(* IEC 61131-3 sources: IEC-63313-ST-Simulator/grammar/src/test/resources/iec61131_structuredtext, 20 files *)

(* ---- type.st ---- *)
TYPE ST_CAN_RXTX :
STRUCT
	uiTXCounter				:	UINT;
	uiRxCounter				:	UINT;
	uiNoOfRxTxMessages		:	UINT;
//	ar_stRxTxMessage		:	ARRAY[0..9] OF ST_CAN_RXTX_MESSAGE;
END_STRUCT;
END_TYPE

TYPE ST_CAN_RXTX_MESSAGE :
STRUCT
	uiLength		:	UINT;
	udCobId			:	UDINT;
//	ar_usiData		:	ARRAY[0..7] OF USINT;
END_STRUCT;
END_TYPE

TYPE ST_GezeFTV :
STRUCT
	bEntriegelt					:	BOOL;
	bVerriegelt					:	BOOL;
	bRunAlarm					:	BOOL;
	bTuerZu						:	BOOL;	// 1/4
	bRueckmeldungVerriegelung	:	BOOL;	// 1/7
	bTuerAlarmZentrale			:	BOOL;	// 2/2
	bKurzzeitfreigabe			:	BOOL;
END_STRUCT;
END_TYPE

(* ---- type_bool_struct.st ---- *)
TYPE
  S_FA_STATUS : STRUCT
    BART_Hand : BOOL := TRUE;
    BART_Auto : BOOL := FALSE;
    Stoerung : BOOL := FALSE;
    Stoer_Quit : BOOL := FALSE;
    NotHalt : BOOL := FALSE;
    Takt : BOOL := FALSE;
  END_STRUCT;
END_TYPE

(* ---- interface.st ---- *)
INTERFACE I_Subject

METHOD Attach : BOOL
VAR_INPUT
	ipObserver		: I_Observer;
END_VAR

METHOD Detach : BOOL
VAR_INPUT
	ipObserver		: I_Observer;
END_VAR

(* ---- function_selection.st ---- *)
FUNCTION SEL : ANY (* binary selection *)
  VAR_INPUT
    G : BOOL;
    IN0 : ANY;
    IN1 : ANY;
  END_VAR
  IF G = 0 THEN
    SEL := IN0; (* selection of upper input *)
  ELSE
    SEL := IN1; (*selection of lower input *)
  END_IF;
END_FUNCTION

(* ---- function_block.st ---- *)
FUNCTION_BLOCK PUBLIC FB_Logger
VAR
  sFilenameExtension : STRING;
END_VAR

// A method starts with a declaration
METHOD PUBLIC Write : STRING
VAR_INPUT
  sMsg : STRING;
END_VAR

// A method declaration is followed by statements that form
// the method's body.
// The next method declaration implicitly terminates the
// preceding method's body!
IF G = 0 THEN
	SEL := 1;
ELSE
	SEL := 2;
END_IF;

/*
sMsg := CONCAT('logger: ', sMsg);
IF (sFilenameExtension = 'txt') THEN
  Write := WriteTxt(sMsg);
ELSIF (sFilenameExtension = 'csv') THEN
  Write := WriteCsv(sMsg);
ELSIF (sFilenameExtension = 'xml') THEN
  Write := WriteXml(sMsg);
END_IF
*/

METHOD CreateErrorLogDB : BOOL
VAR_INPUT
    sDBName : T_MaxString;
END_VAR

CASE nState_CreateDB OF
    0:
    	stDBConfig.sServer := CONCAT(CONCAT(sDBPath, sDBName), '.sdf');
    	stDBConfig.bAuthentification := FALSE;

    	nState_CreateDB := 1;
    1:
        IF fbPLCDBCreate.Database(pDatabaseConfig:= ADR(stDBConfig),
            cbDatabaseConfig:= SIZEOF(stDBConfig),
            bCreateXMLConfig:= FALSE,
            pDBID:= 0) THEN
            ipResultEvt := fbPLCDBCreate.ipTcResult;
            IF fbPLCDBCreate.bError THEN
                nState_CreateDB := 100;
            ELSE
                nState_CreateDB := 2;
            END_IF;
        END_IF;
     2:
        IF fbConfigTcDBSrv.Create(pTcDBSrvConfig:= ADR(stDBConfig),
            cbTcDBSrvConfig:= SIZEOF(stDBConfig), bTemporary:= TRUE,
             pConfigID:= ADR(nDBID) ) THEN
            ipResultEvt := fbConfigTcDBSrv.ipTcResult;
            IF fbConfigTcDBSrv.bError THEN
                nState_CreateDB := 100;
            ELSE
                nState_CreateDB := 3;
            END_IF;
        END_IF;
     3:
     	arrTableColumns[0].sName := 'ID';
        arrTableColumns[0].eType := E_ColumnType.BigInt;
        arrTableColumns[0].nLength := 8;
        arrTableColumns[0].sProperty := 'IDENTITY(1,1)';

        arrTableColumns[1].sName := 'Timestamp';
        arrTableColumns[1].eType := E_ColumnType.DateTime;
        arrTableColumns[1].nLength := 4;

        arrTableColumns[2].sName := 'Severity';
        arrTableColumns[2].eType := E_ColumnType.NVarChar;
        arrTableColumns[2].nLength := 10;

        arrTableColumns[3].sName := 'ErrorCode';
        arrTableColumns[3].eType := E_ColumnType.Integer;
        arrTableColumns[3].nLength := 4;

        arrTableColumns[4].sName := 'Message';
        arrTableColumns[4].eType := E_ColumnType.NVarChar;
        arrTableColumns[4].nLength := 255;

        IF fbPLCDBCreate.Table(hDBID:= nDBID, sTableName:= sTableName,
            pTableCfg:= ADR(arrTableColumns),
            cbTableCfg:= SIZEOF(arrTableColumns)) THEN
            ipResultEvt := fbPLCDBCreate.ipTcResultEvent;
            nState_CreateDB := 100;
        END_IF;
    100:
        IF _SetResultInfo(1033) THEN
            IF NOT bError THEN
                _bHasCreated := TRUE;
            END_IF;

            nState_CreateDB := 0;
        END_IF;
END_CASE;

END_FUNCTION_BLOCK

(* ---- function_block_inout_var.st ---- *)
FUNCTION_BLOCK FNC_BLK

  VAR_IN_OUT
    var_1 : BOOL;
    var_2 : BOOL;
  END_VAR

  VAR_INPUT
    var_3 : UINT;
    var_4 : UINT;
  END_VAR

END_FUNCTION_BLOCK

(* ---- function_block_simple.st ---- *)
FUNCTION_BLOCK FNC_BLK

  VAR_INPUT
    var_1 : BOOL;
  END_VAR

END_FUNCTION_BLOCK

(* ---- large_program.st ---- *)
/**/
TYPE
  S_FA_STATUS : STRUCT
    BART_Hand : BOOL := TRUE;
    BART_Auto : BOOL := FALSE;
    Stoerung : BOOL := FALSE;
    Stoer_Quit : BOOL := FALSE;
    NotHalt : BOOL := FALSE;
    Takt : BOOL := FALSE;
  END_STRUCT;
END_TYPE

FUNCTION_BLOCK AKT_5_2_MV
  VAR_INPUT
    status : S_FA_STATUS;
    Hand_P1 : BOOL;
    Hand_P2 : BOOL;
  END_VAR
  VAR_INPUT
    SEN_P1 : BOOL;
    SEN_P2 : BOOL;
  END_VAR

  VAR_OUTPUT
    s_MV_P2_FF : BOOL;
  END_VAR

  VAR
    SR0 : SR;
  END_VAR
  VAR
    DebugBoolean : BOOL;
    TON0 : TON;
  END_VAR

  VAR CONSTANT
    const_T_Laufzeit_P2 : TIME := T#10s;
  END_VAR

  VAR
    _TMP_AND6_OUT : BOOL;
    _TMP_AND9_OUT : BOOL;
    _TMP_NOT17_OUT : BOOL;
    _TMP_AND15_OUT : BOOL;
  END_VAR

  // compute the control input for Magnetventil Position 2 using a Reset-dominant flip flop
  // and store the result into the out parameter s_MV_P2_FF
  _TMP_AND6_OUT := AND(status.BART_Hand, Hand_P2);
  _TMP_AND9_OUT := AND(status.BART_Hand, Hand_P1);
  SR0(S1 := _TMP_AND6_OUT, R := _TMP_AND9_OUT);
  s_MV_P2_FF := SR0.Q1;

  // Error detection - Laufzeitueberwachung towards Magnetventil Position 2
  _TMP_NOT17_OUT := NOT(SEN_P2);
  _TMP_AND15_OUT := AND(_TMP_NOT17_OUT, Hand_P2);
  TON0(IN := _TMP_AND15_OUT, PT := const_T_Laufzeit_P2);
  DebugBoolean := TON0.Q;

END_FUNCTION_BLOCK

/* We cannot parse functions yet!
FUNCTION FA_SERV : BOOL
  VAR_INPUT
    status : S_FA_STATUS;
    BART_Hand : BOOL;
    BART_Auto : BOOL;
    Stoerung : BOOL;
    Stoer_Quit : BOOL;
    NotHalt : BOOL;
  END_VAR

  status.BART_Hand := BART_Hand;
  status.BART_Auto := BART_Auto;
  status.Stoerung := Stoerung;
  status.Stoer_Quit := Stoer_Quit;
  status.NotHalt := NotHalt;

  FA_SERV := status.BART_Hand;
END_FUNCTION
*/

PROGRAM program0_POU
  VAR
    FA_Start_T_HMI : BOOL;
    FA_Init_T_HMI : BOOL;
    FA_Sonder_T_HMI : BOOL;
    FA_Stop_T_HMI : BOOL;
    FA_BART_Hand_T_HMI : BOOL := TRUE;
    FA_BART_Auto_T_HMI : BOOL;
    FA_BART_Auto_Einzel_T_HMI : BOOL;
    FA_Stoerung_T_HMI : BOOL;
    FA_Stoer_Quit_T_HMI : BOOL;
    FA_NotHalt_T_HMI : BOOL;
    DebugBoolean : BOOL;
  END_VAR
  VAR_EXTERNAL
    global_status : S_FA_STATUS;
  END_VAR
  VAR
    AKT_5_2_MV0 : AKT_5_2_MV;
    Zyl1_T_P1_HMI : BOOL;
    //Zyl1_T_P2_HMI : BOOL := TRUE;
    Zyl1_T_P2_HMI : BOOL := FALSE;
    //Zyl1_T_P2_HMI : BOOL;
    s_MV_P2_FF : BOOL;
    SEN_P1_T_HMI : BOOL := TRUE;
    SEN_P2_T_HMI : BOOL := FALSE;
    _TMP_FA_SERV1_OUT : BOOL;
  END_VAR

  global_status.BART_Hand := FA_BART_Hand_T_HMI;

  //_TMP_FA_SERV1_OUT := FA_SERV(global_status, FA_BART_Hand_T_HMI, FA_BART_Auto_T_HMI, FA_Stoerung_T_HMI, FA_Stoer_Quit_T_HMI, FA_NotHalt_T_HMI);

  DebugBoolean := _TMP_FA_SERV1_OUT;

  AKT_5_2_MV0(
    status := global_status,
    Hand_P1 := Zyl1_T_P1_HMI,
    Hand_P2 := Zyl1_T_P2_HMI,
    SEN_P1 := SEN_P1_T_HMI,
    SEN_P2 := SEN_P2_T_HMI
  );

  s_MV_P2_FF := AKT_5_2_MV0.s_MV_P2_FF;

END_PROGRAM

FUNCTION_BLOCK FA
  VAR
    Status : S_FA_STATUS;
  END_VAR

  Status.Stoerung := TRUE;
END_FUNCTION_BLOCK

/*
FUNCTION_BLOCK SequenctialFunctionChart
  VAR
    RedLight : BOOL;
    OrangeLight : BOOL;
    GreenLight : BOOL;
    Step_0_Active : BOOL := TRUE;
    Step_1_Active : BOOL := FALSE;
    Step_2_Active : BOOL := FALSE;
    TON0 : TON;
    TON1 : TON;
    TON2 : TON;
  END_VAR

  INITIAL_STEP Step0:
    RedLight(N);
    Step_0_Active(N);
    COMPUTE_FUNCTION_BLOCKS(S);
  END_STEP

  ACTION COMPUTE_FUNCTION_BLOCKS:
    TON0(IN := Step_0_Active, PT := T#6s);
    TON1(IN := Step_1_Active, PT := T#6s);
    TON2(IN := Step_2_Active, PT := T#6s);
  END_ACTION

  TRANSITION FROM Step0 TO Step1
    := TON0.Q;
  END_TRANSITION

  STEP Step1:
    GreenLight(N);
    Step_1_Active(N);
  END_STEP

  TRANSITION FROM Step1 TO Step2
    := TON1.Q;
  END_TRANSITION

  STEP Step2:
    OrangeLight(N);
    Step_2_Active(N);
  END_STEP

  TRANSITION FROM Step2 TO Step0
    := TON2.Q;
  END_TRANSITION

END_FUNCTION_BLOCK
*/

CONFIGURATION Config0

  RESOURCE Res0 ON PLC
    VAR_GLOBAL
      global_status : S_FA_STATUS;
    END_VAR
    TASK task0(INTERVAL := T#20ms,PRIORITY := 0);
    PROGRAM instance0 WITH task0 : program0_POU;
  END_RESOURCE

END_CONFIGURATION

(* ---- large_program_2.st ---- *)
TYPE
  S_FA_STATUS : STRUCT
    BART_Hand : BOOL := TRUE;
    BART_Auto : BOOL := FALSE;
    Stoerung : BOOL := FALSE;
    Stoer_Quit : BOOL := FALSE;
    NotHalt : BOOL := FALSE;
    Takt : BOOL := FALSE;
  END_STRUCT;
END_TYPE

FUNCTION_BLOCK AKT_5_2_MV
    /**/
  VAR_IN_OUT
    status : S_FA_STATUS;
  END_VAR

  VAR_INPUT
    //status : S_FA_STATUS;
    Hand_P1 : BOOL;
    Hand_P2 : BOOL;
  END_VAR
  VAR
    SR0 : SR;
  END_VAR
  VAR_OUTPUT
    s_MV_P2_FF : BOOL;
  END_VAR
  VAR
    DebugBoolean : BOOL;
    TON0 : TON;
  END_VAR
  VAR CONSTANT
    const_T_Laufzeit_P2 : TIME := T#10s;
  END_VAR
  VAR_INPUT
    SEN_P1 : BOOL;
    SEN_P2 : BOOL;
  END_VAR
  VAR
    _TMP_AND6_OUT : BOOL;
    _TMP_AND9_OUT : BOOL;
    _TMP_NOT17_OUT : BOOL;
    _TMP_AND15_OUT : BOOL;
  END_VAR

  _TMP_AND6_OUT := AND(status.BART_Hand, Hand_P2);
  _TMP_AND9_OUT := AND(status.BART_Hand, Hand_P1);
  SR0(S1 := _TMP_AND6_OUT, R := _TMP_AND9_OUT);
  s_MV_P2_FF := SR0.Q1;
  _TMP_NOT17_OUT := NOT(SEN_P2);
  _TMP_AND15_OUT := AND(_TMP_NOT17_OUT, Hand_P2);
  TON0(IN := _TMP_AND15_OUT, PT := const_T_Laufzeit_P2);
  status.Stoerung := TON0.Q;
END_FUNCTION_BLOCK

/*
FUNCTION FA_SERV : BOOL
  VAR_INPUT
    status : S_FA_STATUS;
    BART_Hand : BOOL;
    BART_Auto : BOOL;
    Stoerung : BOOL;
    Stoer_Quit : BOOL;
    NotHalt : BOOL;
  END_VAR

  status.BART_Hand := BART_Hand;
  FA_SERV := status.BART_Hand;
  status.BART_Auto := BART_Auto;
  status.Stoerung := Stoerung;
  status.Stoer_Quit := Stoer_Quit;
  status.NotHalt := NotHalt;
END_FUNCTION
*/

PROGRAM program0_POU
  VAR
    FA_Start_T_HMI : BOOL;
    FA_Init_T_HMI : BOOL;
    FA_Sonder_T_HMI : BOOL;
    FA_Stop_T_HMI : BOOL;
    FA_BART_Hand_T_HMI : BOOL := TRUE;
    FA_BART_Auto_T_HMI : BOOL;
    FA_BART_Auto_Einzel_T_HMI : BOOL;
    FA_Stoerung_T_HMI : BOOL;
    FA_Stoer_Quit_T_HMI : BOOL;
    FA_NotHalt_T_HMI : BOOL;
    DebugBoolean : BOOL;
  END_VAR
  VAR_EXTERNAL
    global_status : S_FA_STATUS;
  END_VAR
  VAR
    AKT_5_2_MV0 : AKT_5_2_MV;
    Zyl1_T_P1_HMI : BOOL;
    Zyl1_T_P2_HMI : BOOL;
    s_MV_P2_FF : BOOL;
    SEN_P1_T_HMI : BOOL := TRUE;
    SEN_P2_T_HMI : BOOL := FALSE;
    _TMP_FA_SERV1_OUT : BOOL;
  END_VAR

  global_status.BART_Hand := FA_BART_Hand_T_HMI;
  //_TMP_FA_SERV1_OUT := FA_SERV(global_status, FA_BART_Hand_T_HMI, FA_BART_Auto_T_HMI, FA_Stoerung_T_HMI, FA_Stoer_Quit_T_HMI, FA_NotHalt_T_HMI);
  DebugBoolean := _TMP_FA_SERV1_OUT;
  AKT_5_2_MV0(status := global_status, Hand_P1 := Zyl1_T_P1_HMI, Hand_P2 := Zyl1_T_P2_HMI, SEN_P1 := SEN_P1_T_HMI, SEN_P2 := SEN_P2_T_HMI);
  s_MV_P2_FF := AKT_5_2_MV0.s_MV_P2_FF;
END_PROGRAM

FUNCTION_BLOCK FA
  VAR
    Status : S_FA_STATUS;
  END_VAR

  Status.Stoerung := TRUE;
END_FUNCTION_BLOCK

/*
FUNCTION_BLOCK SequenctialFunctionChart
  VAR
    RedLight : BOOL;
    OrangeLight : BOOL;
    GreenLight : BOOL;
    Step_0_Active : BOOL := TRUE;
    Step_1_Active : BOOL := FALSE;
    Step_2_Active : BOOL := FALSE;
    TON0 : TON;
    TON1 : TON;
    TON2 : TON;
  END_VAR

  INITIAL_STEP Step0:
    RedLight(N);
    Step_0_Active(N);
    COMPUTE_FUNCTION_BLOCKS(S);
  END_STEP

  ACTION COMPUTE_FUNCTION_BLOCKS:
    TON0(IN := Step_0_Active, PT := T#6s);
    TON1(IN := Step_1_Active, PT := T#6s);
    TON2(IN := Step_2_Active, PT := T#6s);
  END_ACTION

  TRANSITION FROM Step0 TO Step1
    := TON0.Q;
  END_TRANSITION

  STEP Step1:
    GreenLight(N);
    Step_1_Active(N);
  END_STEP

  TRANSITION FROM Step1 TO Step2
    := TON1.Q;
  END_TRANSITION

  STEP Step2:
    OrangeLight(N);
    Step_2_Active(N);
  END_STEP

  TRANSITION FROM Step2 TO Step0
    := TON2.Q;
  END_TRANSITION

END_FUNCTION_BLOCK
*/

CONFIGURATION Config0

  RESOURCE Res0 ON PLC
    VAR_GLOBAL
      global_status : S_FA_STATUS;
    END_VAR
    TASK task0(INTERVAL := T#20ms,PRIORITY := 0);
    PROGRAM instance0 WITH task0 : program0_POU;
  END_RESOURCE
END_CONFIGURATION

(* ---- large_program_3.st ---- *)
TYPE
  S_FA_STATUS : STRUCT
    BART_Hand : BOOL := TRUE;
    BART_Auto : BOOL := FALSE;
    Stoerung : BOOL := FALSE;
    Stoer_Quit : BOOL := FALSE;
    NotHalt : BOOL := FALSE;
    Takt : BOOL := FALSE;
  END_STRUCT;
END_TYPE

FUNCTION_BLOCK AKT_5_2_MV
  VAR_IN_OUT
    status : S_FA_STATUS;
  END_VAR
  VAR_INPUT
    Hand_P1 : BOOL;
    Hand_P2 : BOOL;
  END_VAR
  VAR
    SR0 : SR;
  END_VAR
  VAR_OUTPUT
    s_MV_P2_FF : BOOL;
  END_VAR
  VAR
    DebugBoolean : BOOL;
    TON0 : TON;
  END_VAR
  VAR CONSTANT
    const_T_Laufzeit_P2 : TIME := T#10s;
  END_VAR
  VAR_INPUT
    SEN_P1 : BOOL;
    SEN_P2 : BOOL;
  END_VAR
  VAR
    RS0 : RS;
  END_VAR
  VAR_INPUT
    F_LZ_P2 : RS;
  END_VAR
  VAR_OUTPUT
    F_LZ_P3 : BOOL;
  END_VAR
  VAR
    _TMP_AND6_OUT : BOOL;
    _TMP_AND9_OUT : BOOL;
    _TMP_NOT17_OUT : BOOL;
    _TMP_AND15_OUT : BOOL;
  END_VAR

  _TMP_AND6_OUT := AND(status.BART_Hand, Hand_P2);
  _TMP_AND9_OUT := AND(status.BART_Hand, Hand_P1);
  SR0(S1 := _TMP_AND6_OUT, R := _TMP_AND9_OUT);
  s_MV_P2_FF := SR0.Q1;
  _TMP_NOT17_OUT := NOT(SEN_P2);
  _TMP_AND15_OUT := AND(_TMP_NOT17_OUT, Hand_P2);
  TON0(IN := _TMP_AND15_OUT, PT := const_T_Laufzeit_P2);
  RS0(S := TON0.Q);
  F_LZ_P3 := RS0.Q1;
END_FUNCTION_BLOCK
/*
FUNCTION FA_SERV : BOOL
  VAR_INPUT
    status : S_FA_STATUS;
    BART_Hand : BOOL;
    BART_Auto : BOOL;
    Stoerung : BOOL;
    Stoer_Quit : BOOL;
    NotHalt : BOOL;
  END_VAR

  status.BART_Hand := BART_Hand;
  FA_SERV := status.BART_Hand;
  status.BART_Auto := BART_Auto;
  status.Stoerung := Stoerung;
  status.Stoer_Quit := Stoer_Quit;
  status.NotHalt := NotHalt;
END_FUNCTION
*/
PROGRAM program0_POU
  VAR
    FA_Start_T_HMI : BOOL;
    FA_Init_T_HMI : BOOL;
    FA_Sonder_T_HMI : BOOL;
    FA_Stop_T_HMI : BOOL;
    FA_BART_Hand_T_HMI : BOOL := TRUE;
    FA_BART_Auto_T_HMI : BOOL;
    FA_BART_Auto_Einzel_T_HMI : BOOL;
    FA_Stoerung_T_HMI : BOOL;
    FA_Stoer_Quit_T_HMI : BOOL;
    FA_NotHalt_T_HMI : BOOL;
    DebugBoolean : BOOL;
  END_VAR
  VAR_EXTERNAL
    global_status : S_FA_STATUS;
  END_VAR
  VAR
    AKT_5_2_MV0 : AKT_5_2_MV;
    Zyl1_T_P1_HMI : BOOL;
    Zyl1_T_P2_HMI : BOOL;
    s_MV_P2_FF : BOOL;
    SEN_P1_T_HMI : BOOL := TRUE;
    SEN_P2_T_HMI : BOOL := FALSE;
    _TMP_FA_SERV1_OUT : BOOL;
  END_VAR

  global_status.BART_Hand := FA_BART_Hand_T_HMI;
  //_TMP_FA_SERV1_OUT := FA_SERV(global_status, FA_BART_Hand_T_HMI, FA_BART_Auto_T_HMI, FA_Stoerung_T_HMI, FA_Stoer_Quit_T_HMI, FA_NotHalt_T_HMI);
  DebugBoolean := _TMP_FA_SERV1_OUT;
  AKT_5_2_MV0(status := global_status, Hand_P1 := Zyl1_T_P1_HMI, Hand_P2 := Zyl1_T_P2_HMI, SEN_P1 := SEN_P1_T_HMI, SEN_P2 := SEN_P2_T_HMI);
  s_MV_P2_FF := AKT_5_2_MV0.s_MV_P2_FF;
END_PROGRAM

FUNCTION_BLOCK FA
  VAR
    Status : S_FA_STATUS;
  END_VAR

  Status.Stoerung := TRUE;
END_FUNCTION_BLOCK

/*
FUNCTION_BLOCK SequenctialFunctionChart
  VAR
    RedLight : BOOL;
    OrangeLight : BOOL;
    GreenLight : BOOL;
    Step_0_Active : BOOL := TRUE;
    Step_1_Active : BOOL := FALSE;
    Step_2_Active : BOOL := FALSE;
    TON0 : TON;
    TON1 : TON;
    TON2 : TON;
  END_VAR

  INITIAL_STEP Step0:
    RedLight(N);
    Step_0_Active(N);
    COMPUTE_FUNCTION_BLOCKS(S);
  END_STEP

  ACTION COMPUTE_FUNCTION_BLOCKS:
    TON0(IN := Step_0_Active, PT := T#6s);
    TON1(IN := Step_1_Active, PT := T#6s);
    TON2(IN := Step_2_Active, PT := T#6s);
  END_ACTION

  TRANSITION FROM Step0 TO Step1
    := TON0.Q;
  END_TRANSITION

  STEP Step1:
    GreenLight(N);
    Step_1_Active(N);
  END_STEP

  TRANSITION FROM Step1 TO Step2
    := TON1.Q;
  END_TRANSITION

  STEP Step2:
    OrangeLight(N);
    Step_2_Active(N);
  END_STEP

  TRANSITION FROM Step2 TO Step0
    := TON2.Q;
  END_TRANSITION

END_FUNCTION_BLOCK
*/

CONFIGURATION Config0

  RESOURCE Res0 ON PLC
    VAR_GLOBAL
      global_status : S_FA_STATUS;
    END_VAR
    TASK task0(INTERVAL := T#20ms,PRIORITY := 0);
    PROGRAM instance0 WITH task0 : program0_POU;
  END_RESOURCE
END_CONFIGURATION

(* ---- large_program_4.st ---- *)
TYPE
  S_FA_STATUS : STRUCT
    BART_Hand : BOOL := TRUE;
    BART_Auto : BOOL := FALSE;
    Stoerung : BOOL := FALSE;
    Stoer_Quit : BOOL := FALSE;
    NotHalt : BOOL := FALSE;
    Takt : BOOL := FALSE;
  END_STRUCT;
  Diag : STRUCT
    F_Paar_EN : BOOL := TRUE;
    F_LZ_P1_EN : BOOL := TRUE;
    F_LZ_P2_EN : BOOL := TRUE;
    F_LZ_P1_Zeit : TIME;
    F_LZ_P2_Zeit : TIME;
    Stoerung : BOOL := FALSE;
  END_STRUCT;
END_TYPE

FUNCTION_BLOCK AKT_5_2_MV
  VAR_IN_OUT
    status : S_FA_STATUS;
  END_VAR
  VAR_INPUT
    Hand_P1 : BOOL;
    Hand_P2 : BOOL;
  END_VAR
  VAR
    SR0 : SR;
    SR1 : SR;
  END_VAR
  VAR_OUTPUT
    s_MV_P1_FF : BOOL;
    s_MV_P2_FF : BOOL;
  END_VAR
  VAR
    DebugBoolean : BOOL;
    TON0 : TON;
    TON1 : TON;
  END_VAR
  VAR CONSTANT
    const_T_Laufzeit_P2 : TIME := T#10s;
  END_VAR
  VAR_INPUT
    SEN_P1 : BOOL;
    SEN_P2 : BOOL;
  END_VAR
  VAR
    RS0 : RS;
    RS1 : RS;
  END_VAR
  VAR_INPUT
    F_LZ_P2 : RS;
  END_VAR
  VAR_OUTPUT
    F_LZ_P3 : BOOL;
    F_LZ_P4 : BOOL;
  END_VAR
  VAR_IN_OUT
    Diag : Diag;
  END_VAR
  VAR
    _TMP_AND6_OUT : BOOL;
    _TMP_AND9_OUT : BOOL;
    _TMP_NOT17_OUT : BOOL;
    _TMP_AND15_OUT : BOOL;
    _TMP_OR30_OUT : BOOL;
    _TMP_NOT2_OUT : BOOL;
    _TMP_AND19_OUT : BOOL;
    _TMP_AND18_OUT : BOOL;
    _TMP_AND36_OUT : BOOL;
  END_VAR

  _TMP_AND6_OUT := AND(status.BART_Hand, Hand_P2);
  _TMP_AND9_OUT := AND(status.BART_Hand, Hand_P1);
  SR0(S1 := _TMP_AND6_OUT, R := _TMP_AND9_OUT);
  s_MV_P2_FF := SR0.Q1;

  _TMP_NOT17_OUT := NOT(SEN_P2);
  _TMP_AND15_OUT := AND(_TMP_NOT17_OUT, Hand_P2);
  TON0(IN := _TMP_AND15_OUT, PT := const_T_Laufzeit_P2);
  RS0(S := TON0.Q);

  _TMP_NOT2_OUT := NOT(SEN_P1);
  _TMP_AND19_OUT := AND(_TMP_NOT2_OUT, Hand_P1);
  TON1(IN := _TMP_AND19_OUT, PT := const_T_Laufzeit_P2);
  RS1(S := TON1.Q);

  F_LZ_P3 := RS0.Q1;
  _TMP_OR30_OUT := OR(F_LZ_P3, F_LZ_P4);
  Diag.Stoerung := _TMP_OR30_OUT;

  F_LZ_P4 := RS1.Q1;
  _TMP_AND18_OUT := AND(status.BART_Hand, Hand_P1);
  _TMP_AND36_OUT := AND(status.BART_Hand, Hand_P2);
  SR1(S1 := _TMP_AND18_OUT, R := _TMP_AND36_OUT);
  s_MV_P1_FF := SR1.Q1;

END_FUNCTION_BLOCK

/*
FUNCTION FA_SERV : BOOL
  VAR_INPUT
    status : S_FA_STATUS;
    BART_Hand : BOOL;
    BART_Auto : BOOL;
    Stoerung : BOOL;
    Stoer_Quit : BOOL;
    NotHalt : BOOL;
  END_VAR

  status.BART_Hand := BART_Hand;
  FA_SERV := status.BART_Hand;
  status.BART_Auto := BART_Auto;
  status.Stoerung := Stoerung;
  status.Stoer_Quit := Stoer_Quit;
  status.NotHalt := NotHalt;
END_FUNCTION
*/

PROGRAM program0_POU
  VAR
    FA_Start_T_HMI : BOOL;
    FA_Init_T_HMI : BOOL;
    FA_Sonder_T_HMI : BOOL;
    FA_Stop_T_HMI : BOOL;
    FA_BART_Hand_T_HMI : BOOL := TRUE;
    FA_BART_Auto_T_HMI : BOOL;
    FA_BART_Auto_Einzel_T_HMI : BOOL;
    FA_Stoerung_T_HMI : BOOL;
    FA_Stoer_Quit_T_HMI : BOOL;
    FA_NotHalt_T_HMI : BOOL;
    DebugBoolean : BOOL;
  END_VAR
  VAR_EXTERNAL
    global_status : S_FA_STATUS;
  END_VAR
  VAR
    AKT_5_2_MV0 : AKT_5_2_MV;
    Zyl1_T_P1_HMI : BOOL := FALSE;
    Zyl1_T_P2_HMI : BOOL := FALSE;
    s_MV_P2_FF : BOOL;
    SEN_P1_T_HMI : BOOL := TRUE;
    SEN_P2_T_HMI : BOOL := FALSE;
    Diag : Diag;
    _TMP_FA_SERV1_OUT : BOOL;
  END_VAR

  global_status.BART_Hand := FA_BART_Hand_T_HMI;
  //_TMP_FA_SERV1_OUT := FA_SERV(global_status, FA_BART_Hand_T_HMI, FA_BART_Auto_T_HMI, FA_Stoerung_T_HMI, FA_Stoer_Quit_T_HMI, FA_NotHalt_T_HMI);
  //DebugBoolean := _TMP_FA_SERV1_OUT;
  AKT_5_2_MV0(status := global_status, Hand_P1 := Zyl1_T_P1_HMI, Hand_P2 := Zyl1_T_P2_HMI, SEN_P1 := SEN_P1_T_HMI, SEN_P2 := SEN_P2_T_HMI, Diag := Diag);
  s_MV_P2_FF := AKT_5_2_MV0.s_MV_P2_FF;
END_PROGRAM

/*
FUNCTION_BLOCK FA
  VAR
    Status : S_FA_STATUS;
  END_VAR

  Status.Stoerung := TRUE;
END_FUNCTION_BLOCK

FUNCTION_BLOCK SequenctialFunctionChart
  VAR
    RedLight : BOOL;
    OrangeLight : BOOL;
    GreenLight : BOOL;
    Step_0_Active : BOOL := TRUE;
    Step_1_Active : BOOL := FALSE;
    Step_2_Active : BOOL := FALSE;
    TON0 : TON;
    TON1 : TON;
    TON2 : TON;
  END_VAR

  INITIAL_STEP Step0:
    RedLight(N);
    Step_0_Active(N);
    COMPUTE_FUNCTION_BLOCKS(S);
  END_STEP

  ACTION COMPUTE_FUNCTION_BLOCKS:
    TON0(IN := Step_0_Active, PT := T#6s);
    TON1(IN := Step_1_Active, PT := T#6s);
    TON2(IN := Step_2_Active, PT := T#6s);
  END_ACTION

  TRANSITION FROM Step0 TO Step1
    := TON0.Q;
  END_TRANSITION

  STEP Step1:
    GreenLight(N);
    Step_1_Active(N);
  END_STEP

  TRANSITION FROM Step1 TO Step2
    := TON1.Q;
  END_TRANSITION

  STEP Step2:
    OrangeLight(N);
    Step_2_Active(N);
  END_STEP

  TRANSITION FROM Step2 TO Step0
    := TON2.Q;
  END_TRANSITION

END_FUNCTION_BLOCK
*/

CONFIGURATION Config0

  RESOURCE Res0 ON PLC
    VAR_GLOBAL
      global_status : S_FA_STATUS;
    END_VAR
    TASK task0(INTERVAL := T#20ms, PRIORITY := 0);
    PROGRAM instance0 WITH task0 : program0_POU;
  END_RESOURCE
END_CONFIGURATION

(* ---- small_program.st ---- *)
/**/
TYPE
  S_FA_STATUS : STRUCT
    BART_Hand : BOOL := TRUE;
    BART_Auto : BOOL := FALSE;
    Stoerung : BOOL := FALSE;
    Stoer_Quit : BOOL := FALSE;
    NotHalt : BOOL := FALSE;
    Takt : BOOL := FALSE;
  END_STRUCT;
END_TYPE

/**/
FUNCTION_BLOCK AKT_5_2_MV

  VAR_INPUT
    status : S_FA_STATUS;
    Hand_P1 : BOOL;
    Hand_P2 : BOOL;
  END_VAR

  VAR
    SR0 : SR;
  END_VAR

  VAR_OUTPUT
    s_MV_P2_FF : BOOL;
  END_VAR

  VAR
    DebugBoolean : BOOL;
    TON0 : TON;
  END_VAR

  VAR CONSTANT
    const_T_Laufzeit_P2 : TIME := T#10s;
  END_VAR

  VAR_INPUT
    SEN_P1 : BOOL;
    SEN_P2 : BOOL;
  END_VAR

  VAR
    _TMP_AND6_OUT : BOOL;
    _TMP_AND9_OUT : BOOL;
    _TMP_NOT17_OUT : BOOL;
    _TMP_AND15_OUT : BOOL;
  END_VAR

  // OK
  _TMP_AND6_OUT := AND(status.BART_Hand, Hand_P2);

  // OK
  _TMP_AND9_OUT := AND(status.BART_Hand, Hand_P1);

  // OK
  SR0(S1 := _TMP_AND6_OUT, R := _TMP_AND9_OUT);

  // OK
  s_MV_P2_FF := SR0.Q1;

  // OK
  _TMP_NOT17_OUT := NOT(SEN_P2);

  // OK
  _TMP_AND15_OUT := AND(_TMP_NOT17_OUT, Hand_P2);

  // OK
  TON0(IN := _TMP_AND15_OUT, PT := const_T_Laufzeit_P2);

  // OK
  DebugBoolean := TON0.Q;

END_FUNCTION_BLOCK

(* ---- traffic_light.st ---- *)
/**
 * The sequence chart / state machine
 */
FUNCTION_BLOCK SequentialFunctionChart
  VAR
    RedLight : BOOL;
    OrangeLight : BOOL;
    GreenLight : BOOL;
    Step_0_Active : BOOL := TRUE;
    Step_1_Active : BOOL := FALSE;
    Step_2_Active : BOOL := FALSE;
    TON0 : TON;
    TON1 : TON;
    TON2 : TON;
  END_VAR

  INITIAL_STEP Step0:
    RedLight(N);
    Step_0_Active(N);
    COMPUTE_FUNCTION_BLOCKS(S);
  END_STEP

  ACTION COMPUTE_FUNCTION_BLOCKS:
    TON0(IN := Step_0_Active, PT := T#6s);
    TON1(IN := Step_1_Active, PT := T#7s);
    TON2(IN := Step_2_Active, PT := T#8s);
  END_ACTION

  TRANSITION FROM Step0 TO Step1
    := TON0.Q;
  END_TRANSITION

  STEP Step1:
    GreenLight(N);
    Step_1_Active(N);
  END_STEP

  TRANSITION FROM Step1 TO Step2
    := TON1.Q;
  END_TRANSITION

  STEP Step2:
    OrangeLight(N);
    Step_2_Active(N);
  END_STEP

  TRANSITION FROM Step2 TO Step0
    := TON2.Q;
  END_TRANSITION

END_FUNCTION_BLOCK

/**
 * The program
 */
PROGRAM program0_POU
  VAR
    SequentialFunctionChart0 : SequentialFunctionChart;
  END_VAR
  SequentialFunctionChart0();
END_PROGRAM

/**
 * Config
 */
CONFIGURATION Config0
  RESOURCE Res0 ON PLC
    //VAR_GLOBAL
    //  global_status : S_FA_STATUS;
    //END_VAR
    TASK task0(INTERVAL := T#20ms, PRIORITY := 0);
    PROGRAM instance0 WITH task0 : program0_POU;
  END_RESOURCE
END_CONFIGURATION

(* ---- assignment.st ---- *)
PROGRAM program0_POU
    VAR
        FA_Start_T_HMI : BOOL;
    END_VAR

    //test2 := 4 + 14;
    //test2 := 4 - 14;
    //test2 := 4 * 14;
    //test2 := 4 / 14;

    //global_status.BART_Hand := FA_BART_Hand_T_HMI;

    //_TMP_AND15_OUT := AND(_TMP_NOT17_OUT, Hand_P2);

    //_TMP_FA_SERV1_OUT := FA_SERV(global_status, FA_BART_Hand_T_HMI, FA_BART_Auto_T_HMI, FA_Stoerung_T_HMI, FA_Stoer_Quit_T_HMI, FA_NotHalt_T_HMI);

    //FA_SERV(global_status, FA_BART_Hand_T_HMI, FA_BART_Auto_T_HMI, FA_Stoerung_T_HMI, FA_Stoer_Quit_T_HMI, FA_NotHalt_T_HMI);

    AKT_5_2_MV0(status := global_status, Hand_P1 := Zyl1_T_P1_HMI, Hand_P2 := Zyl1_T_P2_HMI, SEN_P1 := SEN_P1_T_HMI, SEN_P2 := SEN_P2_T_HMI);

END_PROGRAM

(* ---- case.st ---- *)
/**/
CASE nState_CreateDB OF
    0:
    	nState_CreateDB := 0;
    1:
    	nState_CreateDB := 1;
    2:
    	nState_CreateDB := 2;
    3:
    	nState_CreateDB := 3;
    100:
    	nState_CreateDB := 100;
    ELSE
    	nState_CreateDB := 101;
END_CASE;

/*
CASE eSeverity OF
    TcEventSeverity.Info:
        stError.sSeverity := 'Info';
    TcEventSeverity.Warning:
        stError.sSeverity := 'Warning';
    TcEventSeverity.Verbose:
        stError.sSeverity := 'Verbose';
    TcEventSeverity.Critical:
        stError.sSeverity := 'Critical';
    TcEventSeverity.Error:
        stError.sSeverity := 'Error';
END_CASE;
*/

(* ---- configuration.st ---- *)
CONFIGURATION Config0
  RESOURCE Res0 ON PLC
    TASK task0(INTERVAL := T#10s, PRIORITY := 12);
    PROGRAM instance0 WITH task0 : stexample;
  END_RESOURCE
END_CONFIGURATION

(* ---- configuration_with_variables.st ---- *)
TYPE
  S_FA_STATUS : STRUCT
    BART_Hand : BOOL := TRUE;
    BART_Auto : BOOL := FALSE;
    Stoerung : BOOL := FALSE;
    Stoer_Quit : BOOL := FALSE;
    NotHalt : BOOL := FALSE;
    Takt : BOOL := FALSE;
  END_STRUCT;
END_TYPE

CONFIGURATION Config0

  RESOURCE Res0 ON PLC
    VAR_GLOBAL
      global_status : S_FA_STATUS;
      //global_status : BOOL;
    END_VAR
    TASK task0(INTERVAL := T#20ms,PRIORITY := 0);
    PROGRAM instance0 WITH task0 : program0_POU;
  END_RESOURCE

END_CONFIGURATION

(* ---- expressions.st ---- *)
PROGRAM expressions

VAR
END_VAR

test := TRUE;

// IF (Tc2_Standard.LEN(STR := MsgFmtString) + LEN(STR := StringArg)) <= MSG_FMT_STRING_MAX_NUMBER_OF_CHARACTERS THEN

IF ((Tc2_Standard.LEN(STR := MsgFmtString) + LEN(STR := StringArg)) <= MSG_FMT_STRING_MAX_NUMBER_OF_CHARACTERS) THEN
	SEL := 1;
END_IF;

(*
IF 1 THEN
	SEL := 1;
END_IF;

IF (1) THEN
	SEL := 1;
END_IF;

IF 1 + (1) THEN
	SEL := 1;
END_IF;

IF (1) + (1) THEN
	SEL := 1;
END_IF;

IF A < 0 THEN
	SEL := 1;
END_IF;

IF A + 1 < 0 THEN
	SEL := 1;
END_IF;

IF A < 0 + 1 THEN
	SEL := 1;
END_IF;

IF A + 1 < 0 + 1 THEN
	SEL := 1;
END_IF;

IF A + 1 + 2 < 0 + 1 + 2 THEN
	SEL := 1;
END_IF;

IF A > 0 THEN
	SEL := 1;
END_IF;

IF A + 1 > 0 THEN
	SEL := 1;
END_IF;

IF A > 0 + 1 THEN
	SEL := 1;
END_IF;

IF A + 1 > 0 + 1 THEN
	SEL := 1;
END_IF;

IF A <= 0 THEN
	SEL := 1;
END_IF;

IF A + 1 <= 0 THEN
	SEL := 1;
END_IF;

IF A <= 0 + 1 THEN
	SEL := 1;
END_IF;

IF A + 1 <= 0 + 1 THEN
	SEL := 1;
END_IF;

IF A >= 0 THEN
	SEL := 1;
END_IF;

IF A + 1 >= 0 THEN
	SEL := 1;
END_IF;

IF A >= 0 + 1 THEN
	SEL := 1;
END_IF;

IF A + 1 >= 0 + 1 THEN
	SEL := 1;
END_IF;

IF (A < 0) THEN
	SEL := 1;
END_IF;

IF (A + 1 < 0) THEN
	SEL := 1;
END_IF;

IF (A < 0 + 1) THEN
	SEL := 1;
END_IF;

IF (A + 1 < 0 + 1) THEN
	SEL := 1;
END_IF;

IF (A > 0) THEN
	SEL := 1;
END_IF;

IF (A + 1 > 0) THEN
	SEL := 1;
END_IF;

IF (A > 0 + 1) THEN
	SEL := 1;
END_IF;

IF (A + 1 > 0 + 1) THEN
	SEL := 1;
END_IF;

IF (A <= 0) THEN
	SEL := 1;
END_IF;

IF (A + 1 <= 0) THEN
	SEL := 1;
END_IF;

IF (A <= 0 + 1) THEN
	SEL := 1;
END_IF;

IF (A + 1 <= 0 + 1) THEN
	SEL := 1;
END_IF;

IF (A >= 0) THEN
	SEL := 1;
END_IF;

IF (A + 1 >= 0) THEN
	SEL := 1;
END_IF;

IF (A >= 0 + 1) THEN
	SEL := 1;
END_IF;

IF (A + 1 >= 0 + 1) THEN
	SEL := 1;
END_IF;

IF (A + 1 + 2 >= 0 + 1 + 2) THEN
	SEL := 1;
END_IF;

IF (A.B >= 1) THEN
	SEL := 1;
END_IF;

IF (1 >= C.D) THEN
	SEL := 1;
END_IF;

IF (A.B >= C.D) THEN
	SEL := 1;
END_IF;
*)

END_PROGRAM

(* ---- program.st ---- *)
PROGRAM M_AIN_2

VAR
END_VAR

//PROGRAM main
/*
VAR
	test: BOOL := TRUE;
	test2: INT := 10;
END_VAR

test := TRUE;
test2 := 14;
*/

(*
VAR
	test: BOOL := TRUE;
	test2: INT := 10;
END_VAR

test := TRUE;
test2 := 14;
*)

VAR
	test: BOOL := FALSE;
	test2: DINT := -12;
	test3: DINT := 0;
END_VAR

test := TRUE;
test2 := -12;
test2 := 4*14;

FOR test2 := 1 TO 10 DO
	test3 := 1;
	//test3 := test3 + 1;
END_FOR;

IF A = 0 THEN
	SEL := 1;
END_IF;

IF G = 0 THEN
	SEL := 1;
ELSE
	SEL := 2;
END_IF;

CASE K OF
 0: MUX := 1;
 1: MUX := 2;
 2: MUX := 3;
END_CASE;

CASE K OF
 0: MUX := 1;
 1: MUX := 2;
 2: MUX := 3;
 ELSE MUX := 4;
END_CASE;

END_PROGRAM

(* ---- self_contained_program.st ---- *)
PROGRAM stexample

  VAR
    x3 : BOOL;
  END_VAR

/**/
  x5 := TRUE;

  x6 := 1 + 2 + 3;
  x7 := 4 + 5 - 6;

/**/
  REPEAT
    x1 := FALSE;
    x2 := FALSE;
  UNTIL x4 = FALSE
  //UNTIL TRUE
  END_REPEAT;

END_PROGRAM

/**/
CONFIGURATION Config0
  RESOURCE Res0 ON PLC
    TASK task0(INTERVAL := T#10s, PRIORITY := 0);
    PROGRAM instance0 WITH task0 : stexample;
  END_RESOURCE
END_CONFIGURATION

// https://www.plcacademy.com/structured-text-tutorial/
